Staubli VAL3: goRemote.pgx

program goRemote()
  local string strGoRemote
begin
  call setSpeed()
  resetMotion()

  strGoRemote = "goRemote "
  strGoRemote = strGoRemote + toString("6.3", pGoRemoteTarget[0].trsf.x)
  strGoRemote = strGoRemote + toString("6.3", pGoRemoteTarget[0].trsf.y)
  strGoRemote = strGoRemote + toString("6.3", pGoRemoteTarget[0].trsf.z)
  strGoRemote = strGoRemote + toString("6.3", pGoRemoteTarget[0].trsf.rx)
  strGoRemote = strGoRemote + toString("6.3", pGoRemoteTarget[0].trsf.ry)
  strGoRemote = strGoRemote + toString("6.3", pGoRemoteTarget[0].trsf.rz)
  call print(strGoRemote)

  movel(pGoRemoteTarget, tTool, mNomSpeed)
  waitEndMove()
end
